// TIA Portal project "4M1" (V16)

(* hardware
DEVICE "S7-1200 station_1"  S7-1200 Station
   slot 0: "Rack_0"  S7-1200 Rack  Rack  V1.0
   slot 1: "PLC_1"  CPU 1212C AC/DC/Rly  6ES7 212-1BE40-0XB0  V4.4
*)

// ===== PLC "PLC_1"  CPU 1212C AC/DC/Rly =====

VAR_GLOBAL   // PLC tag table "Default tag table"
   "START" AT %I0.0 : Bool;
   "STOP" AT %I0.1 : Bool;
   "MOTOR1" AT %Q0.0 : Bool;
   "MOTOR2" AT %Q0.1 : Bool;
   "MOTOR3" AT %Q0.2 : Bool;
   "MOTOR4" AT %Q0.3 : Bool;
   "TM1" AT %M0.0 : Bool;
   "TM2" AT %M0.1 : Bool;
   "X" AT %M0.2 : Bool;
   "TM3" AT %M0.3 : Bool;
   "TM4" AT %M0.4 : Bool;
   "TM5" AT %M0.5 : Bool;
   "CASE1" AT %M0.6 : Bool;
   "CASE2" AT %M0.7 : Bool;
   "CASE3" AT %M1.0 : Bool;
   "CASE4" AT %M1.1 : Bool;
END_VAR

// folder: System blocks/Program resources

DATA_BLOCK "T1"   // DB1
{ S7_Optimized_Access := 'TRUE' }
AUTHOR : Simatic
FAMILY : IEC
NAME : IEC_TMR
VERSION : 1.0
// stored: InstanceOfName IEC_TIMER
"IEC_TIMER"
BEGIN
END_DATA_BLOCK

DATA_BLOCK "T2"   // DB2
{ S7_Optimized_Access := 'TRUE' }
AUTHOR : Simatic
FAMILY : IEC
NAME : IEC_TMR
VERSION : 1.0
// stored: InstanceOfName IEC_TIMER
"IEC_TIMER"
BEGIN
END_DATA_BLOCK

DATA_BLOCK "T3"   // DB3
{ S7_Optimized_Access := 'TRUE' }
AUTHOR : Simatic
FAMILY : IEC
NAME : IEC_TMR
VERSION : 1.0
// stored: InstanceOfName IEC_TIMER
"IEC_TIMER"
BEGIN
END_DATA_BLOCK

DATA_BLOCK "T4"   // DB4
{ S7_Optimized_Access := 'TRUE' }
AUTHOR : Simatic
FAMILY : IEC
NAME : IEC_TMR
VERSION : 1.0
// stored: InstanceOfName IEC_TIMER
"IEC_TIMER"
BEGIN
END_DATA_BLOCK

// folder: (top level)

ORGANIZATION_BLOCK "Main"   // OB1, LAD, ProgramCycle
TITLE = "Main Program Sweep (Cycle)"
{ S7_Optimized_Access := 'TRUE' }
VERSION : 0.1
   VAR_INPUT
      Initial_Call : Bool;   // Initial call of this OB
      Remanence : Bool;   // =True, if remanent data are available
   END_VAR
BEGIN

REGION Network 1
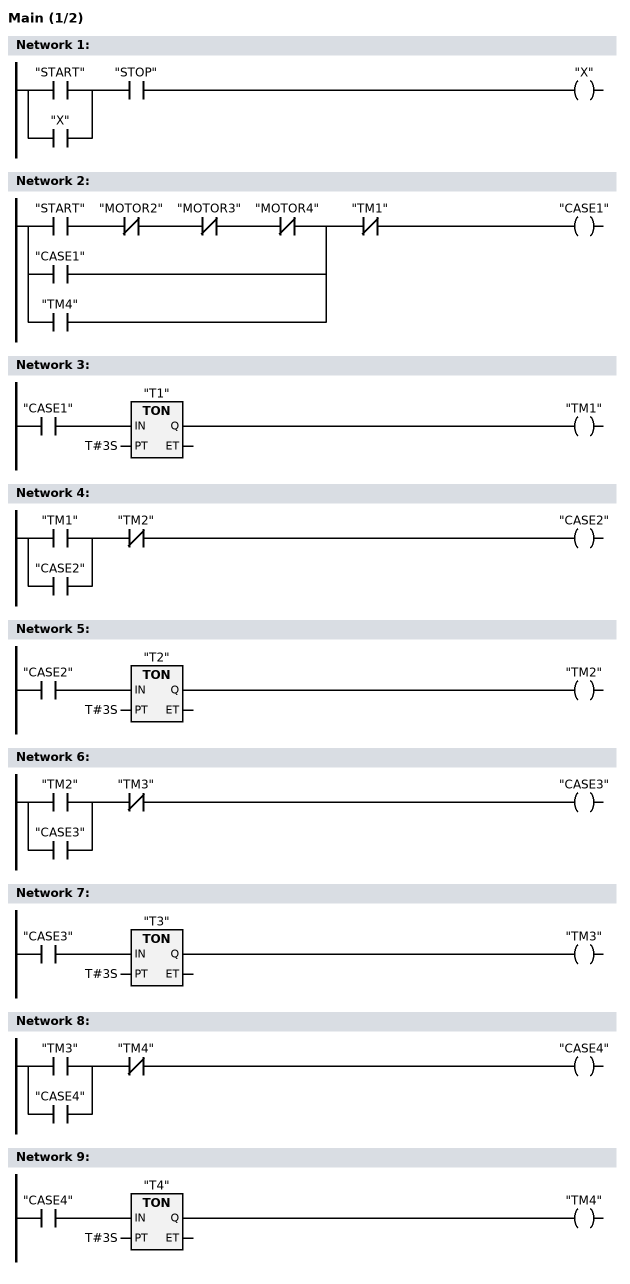
   RUNG wire#powerrail
      Contact( "START" )
      wire#w1
      Contact( "STOP" )
      Coil( "X" )
   END_RUNG
   RUNG wire#powerrail
      Contact( "X" )
   END_RUNG wire#w1
   // the same network as SCL:
   "X" := ("START" OR "X") AND "STOP";
END_REGION

REGION Network 2
   RUNG wire#powerrail
      Contact( "START" )
      I_Contact( "MOTOR2" )
      I_Contact( "MOTOR3" )
      I_Contact( "MOTOR4" )
      wire#w1
      I_Contact( "TM1" )
      Coil( "CASE1" )
   END_RUNG
   RUNG wire#powerrail
      Contact( "CASE1" )
   END_RUNG wire#w1
   RUNG wire#powerrail
      Contact( "TM4" )
   END_RUNG wire#w1
   // the same network as SCL:
   "CASE1" := (("START" AND NOT "MOTOR2" AND NOT "MOTOR3" AND NOT "MOTOR4") OR "CASE1" OR "TM4") AND NOT "TM1";
END_REGION

REGION Network 3
   "T1".TON(IN := "CASE1", PT := T#3S);
   "TM1" := "T1".Q;
END_REGION

REGION Network 4
   RUNG wire#powerrail
      Contact( "TM1" )
      wire#w1
      I_Contact( "TM2" )
      Coil( "CASE2" )
   END_RUNG
   RUNG wire#powerrail
      Contact( "CASE2" )
   END_RUNG wire#w1
   // the same network as SCL:
   "CASE2" := ("TM1" OR "CASE2") AND NOT "TM2";
END_REGION

REGION Network 5
   "T2".TON(IN := "CASE2", PT := T#3S);
   "TM2" := "T2".Q;
END_REGION

REGION Network 6
   RUNG wire#powerrail
      Contact( "TM2" )
      wire#w1
      I_Contact( "TM3" )
      Coil( "CASE3" )
   END_RUNG
   RUNG wire#powerrail
      Contact( "CASE3" )
   END_RUNG wire#w1
   // the same network as SCL:
   "CASE3" := ("TM2" OR "CASE3") AND NOT "TM3";
END_REGION

REGION Network 7
   "T3".TON(IN := "CASE3", PT := T#3S);
   "TM3" := "T3".Q;
END_REGION

REGION Network 8
   RUNG wire#powerrail
      Contact( "TM3" )
      wire#w1
      I_Contact( "TM4" )
      Coil( "CASE4" )
   END_RUNG
   RUNG wire#powerrail
      Contact( "CASE4" )
   END_RUNG wire#w1
   // the same network as SCL:
   "CASE4" := ("TM3" OR "CASE4") AND NOT "TM4";
END_REGION

REGION Network 9
   "T4".TON(IN := "CASE4", PT := T#3S);
   "TM4" := "T4".Q;
END_REGION

REGION Network 10
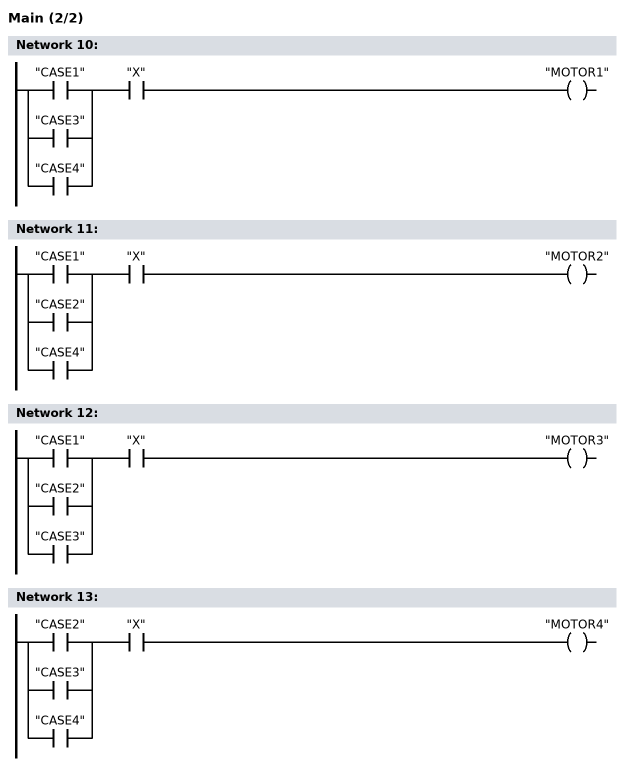
   RUNG wire#powerrail
      Contact( "CASE1" )
      wire#w1
      Contact( "X" )
      Coil( "MOTOR1" )
   END_RUNG
   RUNG wire#powerrail
      Contact( "CASE3" )
   END_RUNG wire#w1
   RUNG wire#powerrail
      Contact( "CASE4" )
   END_RUNG wire#w1
   // the same network as SCL:
   "MOTOR1" := ("CASE1" OR "CASE3" OR "CASE4") AND "X";
END_REGION

REGION Network 11
   RUNG wire#powerrail
      Contact( "CASE1" )
      wire#w1
      Contact( "X" )
      Coil( "MOTOR2" )
   END_RUNG
   RUNG wire#powerrail
      Contact( "CASE2" )
   END_RUNG wire#w1
   RUNG wire#powerrail
      Contact( "CASE4" )
   END_RUNG wire#w1
   // the same network as SCL:
   "MOTOR2" := ("CASE1" OR "CASE2" OR "CASE4") AND "X";
END_REGION

REGION Network 12
   RUNG wire#powerrail
      Contact( "CASE1" )
      wire#w1
      Contact( "X" )
      Coil( "MOTOR3" )
   END_RUNG
   RUNG wire#powerrail
      Contact( "CASE2" )
   END_RUNG wire#w1
   RUNG wire#powerrail
      Contact( "CASE3" )
   END_RUNG wire#w1
   // the same network as SCL:
   "MOTOR3" := ("CASE1" OR "CASE2" OR "CASE3") AND "X";
END_REGION

REGION Network 13
   RUNG wire#powerrail
      Contact( "CASE2" )
      wire#w1
      Contact( "X" )
      Coil( "MOTOR4" )
   END_RUNG
   RUNG wire#powerrail
      Contact( "CASE3" )
   END_RUNG wire#w1
   RUNG wire#powerrail
      Contact( "CASE4" )
   END_RUNG wire#w1
   // the same network as SCL:
   "MOTOR4" := ("CASE2" OR "CASE3" OR "CASE4") AND "X";
END_REGION
END_ORGANIZATION_BLOCK